// TIA Portal V18 export
DATA_BLOCK "CreateDataPair_DB"   // DB1
VERSION : 0.1
// stored: AutoNumber true, InstanceOfName CreateDataPair, InstanceOfType FB
"CreateDataPair"
   // VAR_INPUT
   //    E_Factor : Real;
   //    E_TimeConstant : Real;
   //    E_OffsetY : Real;
   //    P_Form : Real;
   //    P_OffsetX : Real;
   //    P_OffsetY : Real;
   //    S_Length : Real;
   //    S_Amplitude : Real;
   //    S_OffsetX : Real;
   //    S_OffsetY : Real;
   // END_VAR
   // VAR_IN_OUT
   //    TriggerFunction : Int;
   // END_VAR
   // VAR
   //    statIndex { ExternalAccessible := 'False'; ExternalVisible := 'False'; ExternalWritable := 'False'} : Int;
   //    statExponent { ExternalAccessible := 'False'; ExternalVisible := 'False'; ExternalWritable := 'False'} : Real;
   //    statX : Array[0..99] of Real;
   //    statY : Array[0..99] of Real;
   // END_VAR
BEGIN
END_DATA_BLOCK
